PROGRAM MAIN
VAR
END_VAR

END_PROGRAM

(* stored: Version 1.1.0.1, ProductVersion 3.1.4024.6
   POU MAIN: Id {27552b28-ca6c-444c-9236-5c59da3f3bc4}, SpecialFunc None *)
